// TwinCAT 3 PLC project PLC
// ProgramVersion: 3.1.4026.24
// libraries:
//   Tc2_Standard, * (Beckhoff Automation GmbH)
//   Tc2_System, * (Beckhoff Automation GmbH)
//   [Tc3_PlcTestSuite], * (Simmel)
// project tree:
//   / PlcTask.TcTTO
//   POUs/ TestTester.TcPOU, MAIN.TcPOU, SecondTestSuite.TcPOU, TestSuiteOverflow.TcPOU
// real-time tasks:
//   TASK PlcTask: cycle T#10ms, priority 20, ADS port 350

CONFIGURATION PLC
    RESOURCE PLC ON TwinCAT3
        TASK PlcTask(INTERVAL := T#10ms, PRIORITY := 20);
        PROGRAM MAIN WITH PlcTask : MAIN;
    END_RESOURCE
END_CONFIGURATION

// ---- POUs/MAIN.TcPOU
PROGRAM MAIN
VAR
	TestTester		: TestTester;
	ReRun			: BOOL;
	ReRunSingleTest : BOOL;
END_VAR

TestSuite.TestSuiteName := 'My Test Test-Suite';
Test_Counter_AddTwo();
Test_Counter_SubtractTwo();
Test_Bool();
Test_String();
Test_Lreal();
Test_Real();
SecondTestSuite();
TestSuiteOverflow();
IF ReRun THEN
	TestSuite.ReRunTests();
	ReRun := FALSE;
END_IF

IF ReRunSingleTest THEN
	TestSuite.ReRunIndividualTest('MAIN.Test_Counter_AddTwo');
	ReRunSingleTest := FALSE;
END_IF

METHOD Test_Bool
VAR_INST
	Expected : BOOL;
	Actual	 : BOOL;
END_VAR
IF TestSuite.Test(__POUNAME()).ExecuteTest() THEN
	Expected := TRUE;
	Actual	 := TestTester.TestBool;
	TestSuite.Test(__POUNAME()).AssertEqual(Expected, Actual);
END_IF
END_METHOD

METHOD Test_Counter_AddTwo
VAR_INST
	Expected : DINT;
	Actual	 : DINT;
END_VAR
IF TestSuite.Test(__POUNAME()).ExecuteTest() THEN
	Expected := 10;
	Actual	 := TestTester.AddTwo(5, 5);
	TestSuite.Test(__POUNAME()).AssertEqual(Expected, Actual);
END_IF
END_METHOD

METHOD Test_Counter_SubtractTwo
VAR_INST
	Expected : DINT;
	Actual	 : DINT;
END_VAR
IF TestSuite.Test(__POUNAME()).ExecuteTest() THEN
	Expected := 0;
	Actual	 := TestTester.AddTwo(5, -5);
	TestSuite.Test(__POUNAME()).AssertEqual(Expected, Actual);
END_IF
END_METHOD

METHOD Test_Lreal
VAR_INST
	Expected : LREAL;
	Actual	 : LREAL;
END_VAR
IF TestSuite.Test(__POUNAME()).ExecuteTest() THEN
	Expected := 75.75;
	Actual	 := TestTester.TestLReal;
	TestSuite.Test(__POUNAME()).AssertEqual(Expected, Actual, 0.1);
END_IF
END_METHOD

METHOD Test_Real
VAR_INST
	Expected : REAL;
	Actual	 : REAL;
END_VAR
IF TestSuite.Test(__POUNAME()).ExecuteTest() THEN
	Expected := 75.75;
	Actual	 := TestTester.TestLReal;
	TestSuite.Test(__POUNAME()).AssertEqual(Expected, Actual, 0.1);
END_IF
END_METHOD

METHOD Test_String
VAR_INST
	Expected : STRING;
	Actual	 : STRING;
END_VAR
VAR
    SizeString : DINT;
END_VAR
IF TestSuite.Test(__POUNAME()).ExecuteTest() THEN
	Expected := 'TestString';
	Actual	 := TestTester.TestString;
	TestSuite.Test(__POUNAME()).AssertEqual(Expected, Actual);
END_IF
END_METHOD

END_PROGRAM

// ---- POUs/TestTester.TcPOU
FUNCTION_BLOCK TestTester
VAR
END_VAR

METHOD AddTwo : DINT
VAR_INPUT
    In1 : DINT;
    In2 : DINT;
END_VAR
AddTwo := In1 + In2;
END_METHOD

PROPERTY TestBool : BOOL
GET
TestBool := TRUE;
END_GET
SET
END_SET
END_PROPERTY

PROPERTY TestLReal : LREAL
GET
TestLReal := 75.75;
END_GET
SET
END_SET
END_PROPERTY

PROPERTY TestString : STRING
GET
TestString := 'TestString';
END_GET
SET
END_SET
END_PROPERTY

END_FUNCTION_BLOCK

// ---- POUs/SecondTestSuite.TcPOU
PROGRAM SecondTestSuite
VAR
	TestSuite : TestSuite<TestSuiteParameter.MaxTestCount>(ResultFile := JUnitResultFile);
	ReRun	  : BOOL;
END_VAR

TestSuite.TestSuiteName := 'My Second Test-Suite';
Test_OnePlusOne();

IF ReRun THEN
	TestSuite.ReRunTests();
	ReRun := FALSE;
END_IF

METHOD Test_OnePlusOne
VAR_INST
	Expected : DINT;
	Actual	 : DINT;
END_VAR
IF TestSuite.Test(__POUNAME()).ExecuteTest() THEN
	Expected := 2;
	Actual	 := 1 + 1;
	TestSuite.Test(__POUNAME()).AssertEqual(Expected, Actual);
END_IF
END_METHOD

END_PROGRAM

// ---- POUs/TestSuiteOverflow.TcPOU
PROGRAM TestSuiteOverflow
VAR
    TestSuiteOverFlow : TestSuite<2>(ResultFile := JUnitResultFile);
	ReRun		   : BOOL;
END_VAR

TestSuiteOverflow.TestSuiteName := 'Overflow Test-Suite';

Test_TestSuiteOverflow();
Test_TestInstanceOverflow();

IF ReRun THEN
	TestSuiteOverFlow.ReRunTests();
	ReRun := FALSE;
END_IF

METHOD Test_TestInstanceOverflow
VAR_INST
	// Junk instances only used to demonstrate/verify the overflow messages - their XML
	// output is not meant to be inspected by a user, so it is kept out of TEST_Result.xml.
	JunkResultFile : JUnitResultFile<2>('C:\ProgramData\Beckhoff\TwinCAT\3.1\Boot\TEST_InstanceOverflow_Result.xml');
	JunkTestSuite  : TestSuite<2>(ResultFile := JunkResultFile);

	Expected : BOOL;
	Actual	 : BOOL;
END_VAR
VAR
    i : DINT;
END_VAR
IF TestSuite.Test(__POUNAME()).ExecuteTest() THEN
    JunkTestSuite.TestSuiteName := 'Junk Test Instance Overflow';

	// JunkTestSuite<2> only has capacity for 3 tests; a 4th distinct test id forces
	// TestSuite.Test() to hit its "Out of tests" branch and increment TestOverflowCount.
	FOR i := 0 TO 4 DO
		JunkTestSuite.Test(CONCAT('JunkTest_', TO_STRING(i))).ExecuteTest();
	END_FOR

	Expected := TRUE;
	Actual	 := JunkTestSuite.TestOverflowCount > 0;
	TestSuite.Test(__POUNAME()).AssertEqual(Expected, Actual);
END_IF
END_METHOD

METHOD Test_TestSuiteOverflow
VAR_INST
    // Junk instances only used to demonstrate/verify the overflow messages - their XML
	// output is not meant to be inspected by a user, so it is kept out of TEST_Result.xml.
	JunkResultFile : JUnitResultFile<2>('C:\ProgramData\Beckhoff\TwinCAT\3.1\Boot\TEST_SuiteOverflow_Result.xml');
    
	Expected : BOOL;
	Actual	 : BOOL;
END_VAR
VAR
	i : DINT;
END_VAR
IF TestSuite.Test(__POUNAME()).ExecuteTest() THEN
    JunkResultFile.Initialize();

	// JunkResultFile<2> only has capacity for 3 suites; registering 5 distinct suites
	// forces JUnitResultFile.AddTestSuite() to overflow and increment SuiteOverflowCount.
	FOR i := 0 TO 4 DO
		JunkResultFile.AddTestSuite(CONCAT('OverflowSuite_', TO_STRING(i)));
	END_FOR

	Expected := TRUE;
	Actual	 := JunkResultFile.SuiteOverflowCount > 0;
	TestSuite.Test(__POUNAME()).AssertEqual(Expected, Actual);
END_IF
END_METHOD

END_PROGRAM
